{attribute 'qualified_only'}
{attribute 'strict'}
TYPE E_PCM_State :
(
	IDLE,
	MOVEARCHIVE,
	MOVEERROR,
	MOVEKPI,
	GETBYFLAG,
	MOVENEW,
	READ,
	BUILDXMLIMAGE,
	WRITEXMLIMAGE,
	DONE
);
END_TYPE

(* stored: Version 1.1.0.1
   DUT E_PCM_State: Id {d025e04e-245c-4643-8489-074f6d5ef376} *)
